FUNCTION_BLOCK FB_LamparaAsignada_IL
VAR_INPUT
END_VAR
VAR_OUTPUT
END_VAR
VAR
    Lampara AT %Q*: BOOL;
    Pulsador AT %I*: BOOL;
END_VAR

// NETWORK 1
// instruction list
LD      Pulsador
ST      Lampara

END_FUNCTION_BLOCK

(* stored: Version 1.1.0.1, ProductVersion 3.1.4024.12
   POU FB_LamparaAsignada_IL: Id {5a96d4c2-e6d2-4803-a3d9-e8de5affe615}, SpecialFunc None *)
